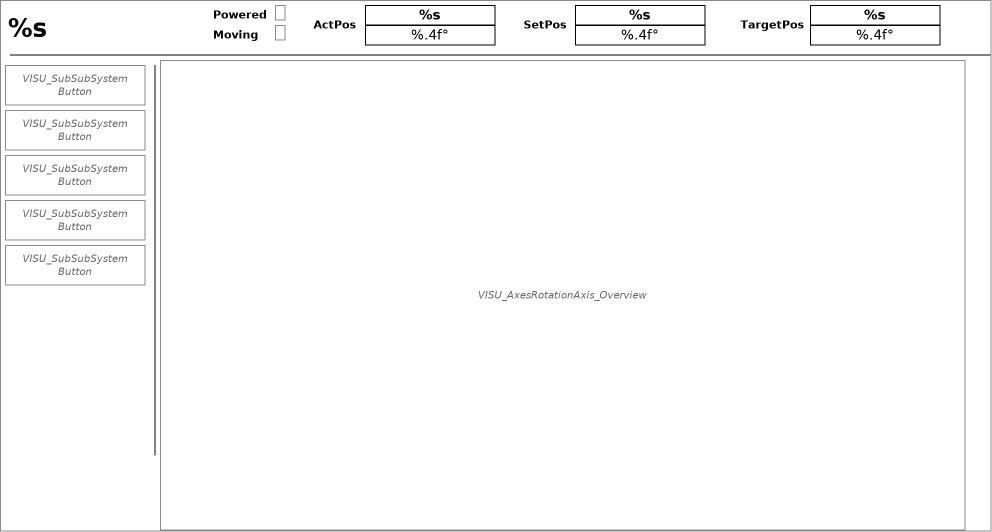
VISUALIZATION VISU_AxesRotationAxis  // 992x532
VAR_IN_OUT
	ref : AxesRotationAxis;
    ref_driveChannel : AX52XXDriveChannel;
    widget : AxesRotationAxisWidget;
END_VAR
    Frame (5,65 140x40)
        shows VISU_SubSubSystemButton(widget := widget.button_overview)
        OnMouseClick: FrameSelectionChange Selection=SelectedFrame=b6fa029b-3640-42a1-bfcc-db8ab31a5104, GlobSel=AssignType=Directly, SelType=Locally
        OnMouseClick: execute { widget.activeTab := AxesRotationAxisTabs.OVERVIEW; }
    Frame (160,60 805x470)
        shows VISU_AxesRotationAxis_Overview(ref := ref, widget := widget)
        shows VISU_AxesRotationAxis_Processes(ref := ref, ref_driveChannel := ref_driveChannel, widget := widget)
        shows VISU_AX522DriveChannel(ref := ref_driveChannel, widget := widget.driveChannel)
        shows VISU_AngularAxis(axis := ref.parts.virtualAxis, widget := widget.virtualAxis)
        shows VISU_AngularAxis(axis := ref.parts.physicalAxis, widget := widget.physicalAxis)
        shows VISU_AxesElevationAxis_AbsoluteEncoder(ref := ref, widget := widget)
        shows VISU_AxesAzimuthAxis_AbsoluteEncoder(ref := ref, widget := widget)
        shows VISU_AxesElevationAxis_Lidas(ref := ref, widget := widget)
        p3523098516: ref
    Line (155,455) (155,65)
    Frame (5,155 140x40)
        shows VISU_SubSubSystemButton(widget := widget.button_driveChannel)
        OnMouseClick: FrameSelectionChange Selection=SelectedFrame=b6fa029b-3640-42a1-bfcc-db8ab31a5104, Selection=2, GlobSel=AssignType=Directly, SelType=Locally
        OnMouseClick: execute { widget.activeTab := AxesRotationAxisTabs.DRIVE_CHANNEL; }
    Frame (5,200 140x40)
        shows VISU_SubSubSystemButton(widget := widget.button_virtualAxis)
        OnMouseClick: FrameSelectionChange Selection=SelectedFrame=b6fa029b-3640-42a1-bfcc-db8ab31a5104, Selection=3, GlobSel=AssignType=Directly, SelType=Locally
        OnMouseClick: execute { widget.activeTab := AxesRotationAxisTabs.VIRTUAL_AXIS; }
    Frame (5,245 140x40)
        shows VISU_SubSubSystemButton(widget := widget.button_physicalAxis)
        OnMouseClick: FrameSelectionChange Selection=SelectedFrame=b6fa029b-3640-42a1-bfcc-db8ab31a5104, Selection=4, GlobSel=AssignType=Directly, SelType=Locally
        OnMouseClick: execute { widget.activeTab := AxesRotationAxisTabs.PHYSICAL_AXIS; }
    Frame (5,110 140x40)
        shows VISU_SubSubSystemButton(widget := widget.button_processes)
        OnMouseClick: FrameSelectionChange Selection=SelectedFrame=b6fa029b-3640-42a1-bfcc-db8ab31a5104, Selection=1, GlobSel=AssignType=Directly, SelType=Locally
        OnMouseClick: execute { widget.activeTab := AxesRotationAxisTabs.PROCESSES; }
    Line (990,55) (10,55)
    Label (305,0 60x50), "ActPos"
    Rectangle (365,5 130x20), "%s", text variable: widget.actPos.dmsString
    Rectangle (365,25 130x20), "%.4f°", text variable: ref.actPos.degrees.value
    Label (515,0 60x50), "SetPos"
    Rectangle (575,5 130x20), "%s", text variable: widget.setPos.dmsString
    Rectangle (575,25 130x20), "%.4f°", text variable: ref.setPos.degrees.value
    Label (735,0 75x50), "TargetPos"
    Rectangle (810,5 130x20), "%s", text variable: widget.targetPos.dmsString
    Rectangle (810,25 130x20), "%.4f°", text variable: ref.targetPos.degrees.value
    Label (210,5 65x20), "Powered"
    Frame (275,5 10x15)
        shows VISU_State_gray_green(state := ref.statuses.poweredStatus.enabled)
    Label (210,25 65x20), "Moving"
    Frame (275,25 10x15)
        shows VISU_State_gray_green(state := ref.parts.physicalAxis.axis_ref.Status.Moving)
    Rectangle (5,5 200x46), "%s", text variable: widget.axisTitle
END_VISUALIZATION

(* stored: Version 1.1.0.1, ProductVersion 3.1.4019.2
   Visu VISU_AxesRotationAxis: Id {4e34055a-3a12-4849-bba3-f901a54f0838} *)
